ABB RobotStudio station: Glider program.rspag

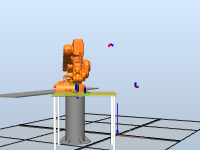
--- station ---
Station E459_norbert (saved by RobotStudio format 3)
Controller IRB140_6kg_0.81m_typeC_1, task T_ROB1: task frame (RAPID world) sits at (10, 680, 720) mm, rotated rx 0 ry 0 rz -30 deg in the station
Controller NorbertEGMVirtuel, task T_ROB1: task frame (RAPID world) sits at (-305, -752, 720) mm, rotated rx 0 ry 0 rz 30 deg in the station
Controller NorbertEGMVirtuel
  mechanical unit ROB_1: Norbert, 6 joints, base frame (0, 0, 0) mm
Controller IRB140_6kg_0.81m_typeC_1
  mechanical unit ROB_1: Rudolf, 6 joints, base frame (0, 0, 0) mm
Layout (positions relative to the parent item):
  - PedestalR [part, from Libraries\Pedestal.rslib] at (10, 680, 0) mm, rotated rx 0 ry 0 rz 150 deg
  - PedestalN [part, from Libraries\Pedestal.rslib] at (-305, -752, 0) mm, rotated rx 0 ry 0 rz -150 deg
  - Windowtable [part]
  - BordN [part, from Libraries\Desk.rslib] at (-421.89, -1050.54, 0) mm, rotated rx 0 ry 0 rz -60 deg
  - BordR [part, from Libraries\Desk.rslib] at (193.4, 1497.66, 0) mm, rotated rx 0 ry 0 rz -120 deg
  - UISpenholder [mechanism, from Libraries\UISpenholder.rslib] at (-60.57, -1074.38, 842.15) mm, rotated rx 179.64 ry 0.98 rz -67.17 deg
  - Norbert [mechanism, from Libraries\IRB140_6_81_C_01.rslib] at (-305, -752, 720) mm, rotated rx 0 ry 0 rz 30 deg; joint values [-1.4454, 0.9396, 0.5122, -0.0137, 0.1371, -2.8775] (rad or m)
  - Rudolf [mechanism, from Libraries\IRB140_6_81_C_01.rslib] at (10, 680, 720) mm, rotated rx 0 ry 0 rz -30 deg; joint values [1.249, 0.6446, -0.2193, 0, 1.1455, 1.249] (rad or m)
Attachment: BordN is attached to PedestalN
Attachment: BordR is attached to PedestalR
Attachment: UISpenholder is attached to Norbert / Link6
Station signals: DI doClose, DI doOpen
Station logic (signal -> signal, property => property):
  NorbertEGMVirtuel.doOpen -> ?.diOpen
  NorbertEGMVirtuel.doClose -> ?.diClose
  ?.doClosed -> NorbertEGMVirtuel.diClosed
Targets, tools, work objects and paths stored in the station and not in the controller backup, written as RAPID:
! task T_ROB1
MODULE EGM_test_UDP
  PROC testAO()
    SetAO ao_Joint1,0;
    SetAO ao_Joint2,0;
    SetAO ao_Joint3,0;
    SetAO ao_Joint4,0;
    SetAO ao_Joint5,0;
    SetAO ao_Joint6,0;
    MoveJ p20,v1000,fine,UISpenholder;
    SetAO ao_MoveX,0;
    SetAO ao_MoveY,0;
    SetAO ao_MoveZ,0;
  ENDPROC
ENDMODULE

! task T_ROB1
MODULE EGM_test_analog
  CONST jointtarget jpos10:=[[0,0,0,0,35,0],[9E9,9E9,9E9,9E9,9E9,9E9]];
  VAR signalao ao_MoveX;
  VAR signalao ao_MoveY;
  VAR signalao ao_MoveZ;
  TASK PERS loaddata load1:=[5,[0,1,0],[1,0,0,0],0,0,0];
  VAR signalao ao_RotX;
  VAR signalao ao_RotY;
  VAR signalao ao_RotZ;
ENDMODULE


--- Backups/IRB140_6kg_0.81m_typeC_1/RAPID/TASK1/PROGMOD/CalibData.mod ---
MODULE CalibData
	TASK PERS wobjdata WorkObj_Bord:=[FALSE,TRUE,"",[[194.800677646,-394.451457857,8],[1,0,0,0]],[[0,0,0],[1,0,0,0]]];


ENDMODULE

--- Backups/IRB140_6kg_0.81m_typeC_1/RAPID/TASK1/PROGMOD/EGMtest.mod ---
MODULE EGMtest
ENDMODULE

--- Backups/NorbertEGMVirtuel/RAPID/TASK1/PROGMOD/CalibData.mod ---
MODULE CalibData
ENDMODULE

--- Backups/NorbertEGMVirtuel/RAPID/TASK1/PROGMOD/EGM_test_UDP.mod ---
MODULE EGM_test_UDP

    VAR egmident egmID1;
    VAR egmstate egmSt1;

    CONST egm_minmax egm_minmax_lin1:=[-1,1]; !in mm
    CONST egm_minmax egm_minmax_rot1:=[-2,2];! in degees
    CONST robtarget p20:=[[34,-499,123],[0.000494947,0.662278052,-0.749217059,-0.007831731],[0,0,-1,0],[9E9,9E9,9E9,9E9,9E9,9E9]];

    PERS tooldata UISpenholder:=[TRUE,[[0,0,114.25],[1,0,0,0]],[1,[-0.095984607,0.082520613,38.69176324],[1,0,0,0],0,0,0]];
    TASK PERS wobjdata wobjBordN:=[FALSE,TRUE,"",[[0,0,0],[1,0,0,0]],[[150,-500,8],[0.707106781,0,0,-0.707106781]]];

    VAR pose posecorTable:=[[150,-500,8],[1,0,0,0]];
    VAR pose posesenTable:=[[0,0,0],[1,0,0,0]];

    PROC main()
        ! Move to start position. Fine point is demanded.
        MoveJ p20,v100,fine,UISpenholder;
        testuc_UDP;
    ENDPROC


    PROC testuc_UDP()
        EGMReset egmID1;
        EGMGetId egmID1;
        egmSt1 := EGMGetState(egmID1);
        TPWrite "EGM state: "\Num := egmSt1;

        IF egmSt1 <= EGM_STATE_CONNECTED THEN
            ! Set up the EGM data source: UdpUc server using device "EGMsensor:"and configuration "default"
            EGMSetupUC ROB_1, egmID1, "default", "EGMSensor:" \pose;
        ENDIF

        !Which program to run
        runEGM;


        IF egmSt1 = EGM_STATE_CONNECTED THEN
            TPWrite "Reset EGM instance egmID1";
            EGMReset egmID1;
        ENDIF
    ENDPROC


        PROC runEGM()
            EGMActPose egmID1\Tool:=UISpenholder \WObj:=wobj0, posecorTable,EGM_FRAME_WOBJ, posesenTable, EGM_FRAME_WOBJ
            \x:=egm_minmax_lin1 \y:=egm_minmax_lin1 \z:=egm_minmax_lin1
            \rx:=egm_minmax_rot1 \ry:=egm_minmax_rot1 \rz:=egm_minmax_rot1\LpFilter:=2\Samplerate:=4\MaxSpeedDeviation:= 1000;

            EGMRunPose egmID1, EGM_STOP_RAMP_DOWN\x \y \z\CondTime:=20 \RampInTime:=0.05\RampOutTime:=0.5;
            egmSt1:=EGMGetState(egmID1);
        ENDPROC

ENDMODULE

--- Backups/NorbertEGMVirtuel/RAPID/TASK1/SYSMOD/LINKEDM.sys ---
%%%
  VERSION:1
  LANGUAGE:ENGLISH
%%%

MODULE LINKEDM (SYSMODULE)

! FOLLOWER
!     Name of electronically linked follower axis used by operator at teach pendent.
      PERS string l_f_axis_name{5}       :=  ["",  "", "", "", ""];

!     Name of the mechanical unit for follower axis.
      PERS string l_f_mecunt_n{5}  :=  ["", "", "", "", ""];

!     Linked follower axis number in the mechanical unit (first axis in mech. unit is number 1).
      PERS num l_f_axis_no{5}      :=  [0,          0,   0,  0,  0];

! MASTER
!     Name of the mechanical unit for linked master axis.
      PERS string l_m_mecunt_n{5} :=  ["", "", "", "", ""];

!     Linked master axis number in the mechanical unit (first axis in mech. unit is number 1).
!     See axis number table in documentation for different master mechanical units.
      PERS num l_m_axis_no{5}     :=  [0,  0,  0,  0,  0];

! POSITION OFFSET
!     The increase of the allowed offset position between the master and follower
!     positions, used when starting AUTO mode. As soon as the offset is decreased
!     the old configurated parameter is used.
!     Example: 3 => the configurated value of allowed offset is increased 3 times.
      PERS num offset_ratio{5}       :=  [10,  10,   10,  10,  10];

! SPEED RATIO
!     Speed_ratio used in AUTO and JOG modes [ very_slow   slow    normal    fast]
!     Value 1 = max allowed manual speed.
      CONST num speed_ratio {20}      := [0.01, 0.01, 0.01, 0.01, 0.01,
                                          0.05, 0.05, 0.05, 0.05, 0.05,
                                          0.20, 0.20, 0.20, 0.20, 0.20,
                                          1.00, 1.00, 1.00, 1.00, 1.00];

! STEP SIZE
!     Displacement position used in JOG mode for each activation of positive or
!     negative movement.                  [very_short    short   normal   long]
!     Unit degees or meter.
      CONST num displacement {20}     := [0.001, 0.001, 0.001, 0.001, 0.001,
                                          0.005, 0.005, 0.005, 0.005, 0.005,
                                          0.020, 0.020, 0.020, 0.020, 0.020,
                                          0.100, 0.100, 0.100, 0.100, 0.100];


!-------------------------------------------------------------
 PROC Linked_m ()
      Linked_m_exe ;
 ENDPROC
ENDMODULE

--- Backups/IRB140_6kg_0.81m_typeC_1/SYSPAR/EIO.cfg ---
EIO:CFG_1.0:5:0::
#
EIO_BUS:

      -Name "Virtual1" -ConnectorID "SIM1"

      -Name "DeviceNet_Lean" -BusType "DNLE" -ConnectorID "PCI1"\
      -ConnectorLabel "DeviceNet Lean"
#
EIO_UNIT_TYPE:

      -Name "Virtual" -VendorName "ABB" -ProductName "Virtual unit"

      -Name "d651_Lean" -BusType "DNLE" -VendorName "ABB Robotics"\
      -ProductName "Combi Unit" -DL_ProductCode 25

      -Name "d652_Lean" -BusType "DNLE" -VendorName "ABB Robotics"\
      -ProductName "24 VDC Unit" -DL_ProductCode 26

      -Name "d653_Lean" -BusType "DNLE" -VendorName "ABB Robotics"\
      -ProductName "Relay Unit" -DL_ProductCode 27

      -Name "AC500_PLC_Lean" -BusType "DNLE" -VendorName "ABB Stotz"\
      -ProductName "AC500 PLC - FPB" -DL_ProductCode 1 -DL_VendorID 760

      -Name "DL_GENERIC" -BusType "DNLE" -DL_ProductCode 3535

      -Name "DL_GENERIC_POLL" -BusType "DNLE" -DL_ProductCode 3535\
      -DL_Pollrate 30

      -Name "d351_Lean" -BusType "DNLE" -VendorName "ABB Robotics"\
      -ProductName "IBS Adapter" -DL_ProductCode 7

      -Name "d378_Lean" -BusType "DNLE" -VendorName "ABB Robotics"\
      -ProductName "CCLink Adapter" -DL_ProductCode 17

      -Name "d377_Lean" -BusType "DNLE" -VendorName "ABB Robotics"\
      -ProductName "Qtracker" -DL_ProductCode 16 -DL_Pollrate 20
#
EIO_UNIT:

      -Name "Qtrack1" -UnitType "d377_Lean" -Bus "DeviceNet_Lean" -DL_Address 10

      -Name "DIGITAL_IO" -UnitType "d652_Lean" -Bus "DeviceNet_Lean"\
      -DL_Address 11
#
EIO_SIGNAL:

      -Name "c1Position" -SignalType "AI" -Unit "Qtrack1" -UnitMap "0-31"\
      -MaxLog 21474.8 -MaxPhys 1 -MaxPhysLimit 1 -MaxBitVal 2147483647\
      -MinLog -21474.8 -MinPhys -1 -MinPhysLimit -1 -MinBitVal -2147483647

      -Name "c1Speed" -SignalType "AI" -Unit "Qtrack1" -UnitMap "32-63"\
      -MaxLog 21474.8 -MaxPhys 1 -MaxPhysLimit 1 -MaxBitVal 2147483647\
      -MinLog -21474.8 -MinPhys -1 -MinPhysLimit -1 -MinBitVal -2147483647

      -Name "c1Connected" -SignalType "DI" -Unit "Qtrack1" -UnitMap "104"

      -Name "c1NullSpeed" -SignalType "DI" -Unit "Qtrack1" -UnitMap "105"

      -Name "c1DReady" -SignalType "DI" -Unit "Qtrack1" -UnitMap "106"

      -Name "c1PassStw" -SignalType "DI" -Unit "Qtrack1" -UnitMap "107"

      -Name "c1NewObjStrobe" -SignalType "DI" -Unit "Qtrack1" -UnitMap "108"

      -Name "c1EncSelected" -SignalType "DI" -Unit "Qtrack1" -UnitMap "109"

      -Name "c1EncAFautlt" -SignalType "DI" -Unit "Qtrack1" -UnitMap "110"

      -Name "c1EncBFautlt" -SignalType "DI" -Unit "Qtrack1" -UnitMap "111"

      -Name "c1Simulating" -SignalType "DI" -Unit "Qtrack1" -UnitMap "112"

      -Name "c1DirOfTravel" -SignalType "DI" -Unit "Qtrack1" -UnitMap "113"

      -Name "c1ScaleEncPuls" -SignalType "DI" -Unit "Qtrack1" -UnitMap "114"

      -Name "c1PowerUpStatus" -SignalType "DI" -Unit "Qtrack1" -UnitMap "83"

      -Name "c1WaitWObj" -SignalType "DO" -Unit "Qtrack1" -UnitMap "0"

      -Name "c1DropWObj" -SignalType "DO" -Unit "Qtrack1" -UnitMap "1"

      -Name "c1Rem1PObj" -SignalType "DO" -Unit "Qtrack1" -UnitMap "2"

      -Name "c1RemAllPObj" -SignalType "DO" -Unit "Qtrack1" -UnitMap "3"

      -Name "c1EncSelect" -SignalType "DO" -Unit "Qtrack1" -UnitMap "4"

      -Name "c1SoftSyncSig" -SignalType "DO" -Unit "Qtrack1" -UnitMap "5"

      -Name "c1SoftCheckSig" -SignalType "DO" -Unit "Qtrack1" -UnitMap "6"

      -Name "c1SimMode" -SignalType "DO" -Unit "Qtrack1" -UnitMap "7"

      -Name "c1CntToEncStr" -SignalType "DO" -Unit "Qtrack1" -UnitMap "40"

      -Name "c1ForceJob" -SignalType "DO" -Unit "Qtrack1" -UnitMap "41"

      -Name "c1PosInJobQ" -SignalType "DO" -Unit "Qtrack1" -UnitMap "42"

      -Name "c1ObjectsInQ" -SignalType "GI" -Unit "Qtrack1" -UnitMap "64-71"

      -Name "c1CntFromEnc1" -SignalType "GI" -Unit "Qtrack1" -UnitMap "72-87"

      -Name "c1CntFromEnc2" -SignalType "GI" -Unit "Qtrack1" -UnitMap "88-103"

      -Name "c1DTimestamp" -SignalType "GI" -Unit "Qtrack1" -UnitMap "120-151"

      -Name "c1CntToEnc1" -SignalType "GO" -Unit "Qtrack1" -UnitMap "8-23"

      -Name "c1CntToEnc2" -SignalType "GO" -Unit "Qtrack1" -UnitMap "24-39"

      -Name "GruppeUt" -SignalType "GO" -Unit "DIGITAL_IO" -UnitMap "0-7"\
      -Access "Default"

      -Name "GruppeInn" -SignalType "GI" -Unit "DIGITAL_IO" -UnitMap "0-7"\
      -Access "Default"

      -Name "LukkeGriper" -SignalType "DO" -Unit "DIGITAL_IO"\
      -SignalLabel "Lukke Griper" -UnitMap "9"

      -Name "Apnegriper" -SignalType "DO" -Unit "DIGITAL_IO"\
      -SignalLabel "Åpne griper" -UnitMap "8"
#
EIO_COMMAND:

      -Unit "Qtrack1" -CommandType "CountsPerMeter" -Value "10000.0"

      -Unit "Qtrack1" -CommandType "SyncSeparation" -Value "0.005"

      -Unit "Qtrack1" -CommandType "QueueTrckDist" -Value "0.0"

      -Unit "Qtrack1" -CommandType "StartWinWidth" -Value "10.0"

      -Unit "Qtrack1" -CommandType "IIRFPeriod" -Value "0.02"

      -Unit "Qtrack1" -CommandType "IIRFNoOfPoles" -Value "2"

      -Unit "Qtrack1" -CommandType "IIRFNoOfZeroes" -Value "0"

      -Unit "Qtrack1" -CommandType "IIRFXfrmMetPol" -Value "1"

      -Unit "Qtrack1" -CommandType "IIRFXfrmMetZero" -Value "1"

      -Unit "Qtrack1" -CommandType "IIRFFZ" -Value "0.0"

      -Unit "Qtrack1" -CommandType "IIRFDZ" -Value "0.0"

      -Unit "Qtrack1" -CommandType "IIRFFP" -Value "2.0"

      -Unit "Qtrack1" -CommandType "IIRFDP" -Value "0.707"

      -Unit "Qtrack1" -CommandType "IIRFGain" -Value "1.0"

      -Unit "Qtrack1" -CommandType "FIRFLength" -Value "0"

      -Unit "Qtrack1" -CommandType "FIRFB0" -Value "0.0"

      -Unit "Qtrack1" -CommandType "FIRFB1" -Value "0.0"

      -Unit "Qtrack1" -CommandType "AutoBackup" -Value "1"

      -Unit "Qtrack1" -CommandType "SimulationVel" -Value "0.100"

      -Unit "Qtrack1" -CommandType "ScalingFactor" -Value "100.0"

      -Unit "Qtrack1" -CommandType "CheckPointDist" -Value "0.0"

      -Unit "Qtrack1" -CommandType "CheckPWinWidth" -Value "0.0"
#
EIO_COMMAND_TYPE:

      -Name "StationNo_L" -UnitType "d378_Lean" -DefValue "1" -OrderNr 1\
      -DL_Path "6,20 68 24 01 30 01,C6,1"

      -Name "BaudRate_L" -UnitType "d378_Lean" -DefValue "0" -OrderNr 2\
      -DL_Path "6,20 68 24 01 30 02,C6,1"

      -Name "OccStat_L" -UnitType "d378_Lean" -DefValue "1" -OrderNr 3\
      -DL_Path "6,20 68 24 01 30 03,C6,1"

      -Name "BasicIO_L" -UnitType "d378_Lean" -DefValue "0" -OrderNr 4\
      -DL_Path "6,20 68 24 01 30 04,C1,1"

      -Name "D378reset_L" -UnitType "d378_Lean" -DefValue "0" -OrderNr 5\
      -DL_Path "4,20 01 24 01,C1,1" -DL_Service 5

      -Name "DataWidth_L" -UnitType "d351_Lean" -DefValue "3" -OrderNr 1\
      -DL_Path "6,20 65 24 01 30 01,C6,1"

      -Name "D351reset_L" -UnitType "d351_Lean" -DefValue "0" -OrderNr 2\
      -DL_Path "4,20 01 24 01,C1,1" -DL_Service 5

      -Name "CountsPerMeter" -UnitType "d377_Lean" -DefValue "10000.0"\
      -OrderNr 2 -DL_Path "6,20 66 24 01 30 01,CA,4"

      -Name "SyncSeparation" -UnitType "d377_Lean" -DefValue "0.1" -OrderNr 3\
      -DL_Path "6,20 66 24 01 30 02,CA,4"

      -Name "QueueTrckDist" -UnitType "d377_Lean" -DefValue "0.0" -OrderNr 4\
      -DL_Path "6,20 66 24 01 30 03,CA,4"

      -Name "StartWinWidth" -UnitType "d377_Lean" -DefValue "0.5" -OrderNr 5\
      -DL_Path "6,20 66 24 01 30 04,CA,4"

      -Name "AutoBackup" -UnitType "d377_Lean" -DefValue "1" -OrderNr 6\
      -DL_Path "6,20 66 24 01 30 12,C1,1"

      -Name "SimulationVel" -UnitType "d377_Lean" -DefValue "0.1" -OrderNr 7\
      -DL_Path "6,20 66 24 01 30 13,CA,4"

      -Name "ScalingFactor" -UnitType "d377_Lean" -DefValue "100" -OrderNr 8\
      -DL_Path "6,20 66 24 01 30 14,CA,4"

      -Name "CheckPointDist" -UnitType "d377_Lean" -DefValue "0.0" -OrderNr 9\
      -DL_Path "6,20 66 24 01 30 15,CA,4"

      -Name "CheckPWinWidth" -UnitType "d377_Lean" -DefValue "0.0" -OrderNr 10\
      -DL_Path "6,20 66 24 01 30 16,CA,4"

      -Name "IIRFPeriod" -UnitType "d377_Lean" -DefValue "0.02" -OrderNr 11\
      -DL_Path "6,20 66 24 01 30 05,CA,4"

      -Name "IIRFNoOfPoles" -UnitType "d377_Lean" -DefValue "2" -OrderNr 12\
      -DL_Path "6,20 66 24 01 30 06,C6,1"

      -Name "IIRFNoOfZeroes" -UnitType "d377_Lean" -DefValue "0" -OrderNr 13\
      -DL_Path "6,20 66 24 01 30 07,C6,1"

      -Name "IIRFXfrmMetPol" -UnitType "d377_Lean" -DefValue "1" -OrderNr 14\
      -DL_Path "6,20 66 24 01 30 08,C6,1"

      -Name "IIRFXfrmMetZero" -UnitType "d377_Lean" -DefValue "1" -OrderNr 15\
      -DL_Path "6,20 66 24 01 30 09,C6,1"

      -Name "IIRFFZ" -UnitType "d377_Lean" -DefValue "0.0" -OrderNr 16\
      -DL_Path "6,20 66 24 01 30 0A,CA,4"

      -Name "IIRFDZ" -UnitType "d377_Lean" -DefValue "0.0" -OrderNr 17\
      -DL_Path "6,20 66 24 01 30 0B,CA,4"

      -Name "IIRFFP" -UnitType "d377_Lean" -DefValue "2.0" -OrderNr 18\
      -DL_Path "6,20 66 24 01 30 0C,CA,4"

      -Name "IIRFDP" -UnitType "d377_Lean" -DefValue "0.707" -OrderNr 19\
      -DL_Path "6,20 66 24 01 30 0D,CA,4"

      -Name "IIRFGain" -UnitType "d377_Lean" -DefValue "1.0" -OrderNr 20\
      -DL_Path "6,20 66 24 01 30 0E,CA,4"

      -Name "FIRFLength" -UnitType "d377_Lean" -DefValue "1" -OrderNr 21\
      -DL_Path "6,20 66 24 01 30 0F,C6,1"

      -Name "FIRFB0" -UnitType "d377_Lean" -DefValue "0.0" -OrderNr 22\
      -DL_Path "6,20 66 24 01 30 10,CA,4"

      -Name "FIRFB1" -UnitType "d377_Lean" -DefValue "0.0" -OrderNr 23\
      -DL_Path "6,20 66 24 01 30 11,CA,4"

      -Name "TimeKeeperInit" -UnitType "d377_Lean" -DefValue "0" -OrderNr 1\
      -DL_Path "6,20 68 24 01 30 01,C1,1"
#
EIO_ACCESS:

      -Name "All" -Rapid  -LocalManual  -LocalAuto  -RemoteManual  -RemoteAuto

--- Backups/NorbertEGMVirtuel/SYSPAR/EIO.cfg ---
EIO:CFG_1.0:6:1::
#
INDUSTRIAL_NETWORK:

      -Name "DeviceNet" -Label "DeviceNet Master/Slave Network" -Address "2"

      -Name "DeviceNet_Anybus" -Label "DeviceNet Anybus Network" -Address "20"
#
DEVICENET_DEVICE:

      -Name "Qtrack1" -Simulated  -VendorName "ABB Robotics"\
      -ProductName "Qtracker" -Address 15 -ProductCode 16 -DeviceType 100\
      -PollRate 20 -OutputSize 6 -InputSize 19

      -Name "DIGITAL_IO" -VendorName "ABB Robotics"\
      -ProductName "24 VDC I/O Device" -Label "DSQC 652 24 VDC I/O Device"\
      -Address 11 -ProductCode 26 -DeviceType 7 -ConnectionType "COS"\
      -OutputSize 2 -InputSize 2
#
DEVICENET_DEVICE_TEMPLATE:

      -Name "d377B" -VendorName "ABB Robotics" -ProductName "Qtracker"\
      -Label "DSQC 377B Queue Tracker" -ProductCode 16 -DeviceType 100\
      -PollRate 20 -OutputSize 6 -InputSize 19
#
DEVICENET_COMMAND:

      -Name "CountsPerMeter1" -Device "Qtrack1" -OrderNr 2\
      -Path "6,20 66 24 01 30 01,CA,4" -Value "20000.0"

      -Name "SyncSeparation1" -Device "Qtrack1" -OrderNr 3\
      -Path "6,20 66 24 01 30 02,CA,4" -Value "0.005"

      -Name "QueueTrckDist1" -Device "Qtrack1" -OrderNr 4\
      -Path "6,20 66 24 01 30 03,CA,4" -Value "0.0"

      -Name "StartWinWidth1" -Device "Qtrack1" -OrderNr 5\
      -Path "6,20 66 24 01 30 04,CA,4" -Value "10.0"

      -Name "AutoBackup1" -Device "Qtrack1" -OrderNr 6\
      -Path "6,20 66 24 01 30 12,C1,1" -Value "1"

      -Name "SimulationVel1" -Device "Qtrack1" -OrderNr 7\
      -Path "6,20 66 24 01 30 13,CA,4" -Value "0.100"

      -Name "ScalingFactor1" -Device "Qtrack1" -OrderNr 8\
      -Path "6,20 66 24 01 30 14,CA,4" -Value "2000.0"

      -Name "CheckPointDist1" -Device "Qtrack1" -OrderNr 9\
      -Path "6,20 66 24 01 30 15,CA,4" -Value "0.0"

      -Name "CheckPWinWidth1" -Device "Qtrack1" -OrderNr 10\
      -Path "6,20 66 24 01 30 16,CA,4" -Value "0.0"

      -Name "IIRFPeriod1" -Device "Qtrack1" -OrderNr 11\
      -Path "6,20 66 24 01 30 05,CA,4" -Value "0.02"

      -Name "IIRFNoOfPoles1" -Device "Qtrack1" -OrderNr 12\
      -Path "6,20 66 24 01 30 06,C6,1" -Value "2"

      -Name "IIRFNoOfZeroes1" -Device "Qtrack1" -OrderNr 13\
      -Path "6,20 66 24 01 30 07,C6,1" -Value "0"

      -Name "IIRFXfrmMetPol1" -Device "Qtrack1" -OrderNr 14\
      -Path "6,20 66 24 01 30 08,C6,1" -Value "1"

      -Name "IIRFXfrmMetZero1" -Device "Qtrack1" -OrderNr 15\
      -Path "6,20 66 24 01 30 09,C6,1" -Value "1"

      -Name "IIRFFZ1" -Device "Qtrack1" -OrderNr 16\
      -Path "6,20 66 24 01 30 0A,CA,4" -Value "0.0"

      -Name "IIRFDZ1" -Device "Qtrack1" -OrderNr 17\
      -Path "6,20 66 24 01 30 0B,CA,4" -Value "0.0"

      -Name "IIRFFP1" -Device "Qtrack1" -OrderNr 18\
      -Path "6,20 66 24 01 30 0C,CA,4" -Value "2.0"

      -Name "IIRFDP1" -Device "Qtrack1" -OrderNr 19\
      -Path "6,20 66 24 01 30 0D,CA,4" -Value "0.707"

      -Name "IIRFGain1" -Device "Qtrack1" -OrderNr 20\
      -Path "6,20 66 24 01 30 0E,CA,4" -Value "1.0"

      -Name "FIRFLength1" -Device "Qtrack1" -OrderNr 21\
      -Path "6,20 66 24 01 30 0F,C6,1" -Value "0"

      -Name "FIRFB01" -Device "Qtrack1" -OrderNr 22\
      -Path "6,20 66 24 01 30 10,CA,4" -Value "0.0"

      -Name "FIRFB11" -Device "Qtrack1" -OrderNr 23\
      -Path "6,20 66 24 01 30 11,CA,4" -Value "0.0"
#
DEVICENET_INTERNAL_DEVICE:

      -Name "DN_Internal_Device" -VendorName "ABB Robotics"\
      -ProductName "DeviceNet Internal Slave Device"
#
DEVICENET_INTERNAL_ANYBUS_DEVICE:

      -Name "DN_Internal_Anybus" -VendorName "ABB Robotics"\
      -ProductName "DeviceNet Internal Anybus Slave Device"
#
EIO_SIGNAL:

      -Name "c1Position" -SignalType "AI" -Device "Qtrack1" -DeviceMap "0-31"\
      -MaxLog 21474.8 -MaxPhys 1 -MaxPhysLimit 1 -MaxBitVal 2147483647\
      -MinLog -21474.8 -MinPhys -1 -MinPhysLimit -1 -MinBitVal -2147483647

      -Name "c1Speed" -SignalType "AI" -Device "Qtrack1" -DeviceMap "32-63"\
      -MaxLog 21474.8 -MaxPhys 1 -MaxPhysLimit 1 -MaxBitVal 2147483647\
      -MinLog -21474.8 -MinPhys -1 -MinPhysLimit -1 -MinBitVal -2147483647

      -Name "c1Connected" -SignalType "DI" -Device "Qtrack1" -DeviceMap "104"

      -Name "c1NullSpeed" -SignalType "DI" -Device "Qtrack1" -DeviceMap "105"

      -Name "c1DReady" -SignalType "DI" -Device "Qtrack1" -DeviceMap "106"

      -Name "c1PassStw" -SignalType "DI" -Device "Qtrack1" -DeviceMap "107"

      -Name "c1NewObjStrobe" -SignalType "DI" -Device "Qtrack1" -DeviceMap "108"

      -Name "c1EncSelected" -SignalType "DI" -Device "Qtrack1" -DeviceMap "109"

      -Name "c1EncAFautlt" -SignalType "DI" -Device "Qtrack1" -DeviceMap "110"

      -Name "c1EncBFautlt" -SignalType "DI" -Device "Qtrack1" -DeviceMap "111"

      -Name "c1Simulating" -SignalType "DI" -Device "Qtrack1" -DeviceMap "112"

      -Name "c1DirOfTravel" -SignalType "DI" -Device "Qtrack1" -DeviceMap "113"

      -Name "c1ScaleEncPuls" -SignalType "DI" -Device "Qtrack1" -DeviceMap "114"

      -Name "c1PowerUpStatus" -SignalType "DI" -Device "Qtrack1" -DeviceMap "83"

      -Name "c1WaitWObj" -SignalType "DO" -Device "Qtrack1" -DeviceMap "0"

      -Name "c1DropWObj" -SignalType "DO" -Device "Qtrack1" -DeviceMap "1"

      -Name "c1Rem1PObj" -SignalType "DO" -Device "Qtrack1" -DeviceMap "2"

      -Name "c1RemAllPObj" -SignalType "DO" -Device "Qtrack1" -DeviceMap "3"

      -Name "c1EncSelect" -SignalType "DO" -Device "Qtrack1" -DeviceMap "4"

      -Name "c1SoftSyncSig" -SignalType "DO" -Device "Qtrack1" -DeviceMap "5"

      -Name "c1SoftCheckSig" -SignalType "DO" -Device "Qtrack1" -DeviceMap "6"

      -Name "c1SimMode" -SignalType "DO" -Device "Qtrack1" -DeviceMap "7"

      -Name "c1CntToEncStr" -SignalType "DO" -Device "Qtrack1" -DeviceMap "40"

      -Name "c1ForceJob" -SignalType "DO" -Device "Qtrack1" -DeviceMap "41"

      -Name "c1PosInJobQ" -SignalType "DO" -Device "Qtrack1" -DeviceMap "42"

      -Name "c1ObjectsInQ" -SignalType "GI" -Device "Qtrack1" -DeviceMap "64-71"

      -Name "c1CntFromEnc" -SignalType "GI" -Device "Qtrack1"\
      -DeviceMap "72-103"

      -Name "c1DTimestamp" -SignalType "GI" -Device "Qtrack1"\
      -DeviceMap "120-151"

      -Name "c1CntToEnc" -SignalType "GO" -Device "Qtrack1" -DeviceMap "8-39"

      -Name "doGripOpen" -SignalType "DO" -Device "DIGITAL_IO"\
      -Label "Pneumatic gripper OPEN" -DeviceMap "9"

      -Name "doGripClose" -SignalType "DO" -Device "DIGITAL_IO"\
      -Label "Pneumatic gripper CLOSE" -DeviceMap "8"

      -Name "ao_Joint1" -SignalType "AO" -Device "Qtrack1" -DeviceMap "16-31"\
      -Access "All" -MaxLog 21474.8 -MaxPhys 500 -MaxPhysLimit 500\
      -MaxBitVal 32767 -MinLog -21474.8 -MinPhys -500 -MinPhysLimit -500\
      -MinBitVal -32767

      -Name "ao_Joint2" -SignalType "AO" -Device "Qtrack1" -DeviceMap "32-47"\
      -MaxLog 21474.8 -MaxPhys 500 -MaxPhysLimit 500 -MaxBitVal 32767\
      -MinLog -21474.8 -MinPhys -500 -MinPhysLimit -500 -MinBitVal -32767

      -Name "ao_Joint3" -SignalType "AO" -Device "Qtrack1" -DeviceMap "48-63"\
      -MaxLog 21474.8 -MaxPhys 500 -MaxPhysLimit 500 -MaxBitVal 32767\
      -MinLog -21474.8 -MinPhys -500 -MinPhysLimit -500 -MinBitVal -32767

      -Name "ao_Joint6" -SignalType "AO" -Device "Qtrack1" -DeviceMap "96-111"\
      -MaxLog 21474.8 -MaxPhys 500 -MaxPhysLimit 500 -MaxBitVal 32767\
      -MinLog -21474.8 -MinPhys -500 -MinPhysLimit -500 -MinBitVal -32767

      -Name "ao_Joint5" -SignalType "AO" -Device "Qtrack1" -DeviceMap "80-95"\
      -MaxLog 21474.8 -MaxPhys 500 -MaxPhysLimit 500 -MaxBitVal 32767\
      -MinLog -21474.8 -MinPhys -500 -MinPhysLimit -500 -MinBitVal -32767

      -Name "ao_Joint4" -SignalType "AO" -Device "Qtrack1" -DeviceMap "64-79"\
      -MaxLog 21474.8 -MaxPhys 500 -MaxPhysLimit 500 -MaxBitVal 32767\
      -MinLog -21474.8 -MinPhys -500 -MinPhysLimit -500 -MinBitVal -32767

      -Name "ao_MoveX" -SignalType "AO" -Device "Qtrack1" -DeviceMap "112-127"\
      -MaxLog 2147.8 -MaxPhys 500 -MaxPhysLimit 500 -MaxBitVal 32767\
      -MinLog -2147.8 -MinPhys -500 -MinPhysLimit -500 -MinBitVal -32767

      -Name "ao_MoveY" -SignalType "AO" -Device "Qtrack1" -DeviceMap "128-143"\
      -MaxLog 21474.8 -MaxPhys 500 -MaxPhysLimit 500 -MaxBitVal 32767\
      -MinLog -21474.8 -MinPhys -500 -MinPhysLimit -500 -MinBitVal -32767

      -Name "ao_MoveZ" -SignalType "AO" -Device "Qtrack1" -DeviceMap "144-159"\
      -MaxLog 21474.8 -MaxPhys 500 -MaxPhysLimit 500 -MaxBitVal 32767\
      -MinLog -21474.8 -MinPhys -500 -MinPhysLimit -500 -MinBitVal -32767

      -Name "ao_RotX" -SignalType "AO" -Device "Qtrack1" -DeviceMap "160-175"\
      -MaxLog 21474.8 -MaxPhys 500 -MaxPhysLimit 500 -MaxBitVal 32767\
      -MinLog -21474.8 -MinPhys -500 -MinPhysLimit -500 -MinBitVal -32767

      -Name "ao_RotY" -SignalType "AO" -Device "Qtrack1" -DeviceMap "176-191"\
      -MaxLog 21474.8 -MaxPhys 500 -MaxPhysLimit 500 -MaxBitVal 32767\
      -MinLog -21474.8 -MinPhys -500 -MinPhysLimit -500 -MinBitVal -32767

      -Name "ao_RotZ" -SignalType "AO" -Device "Qtrack1" -DeviceMap "192-207"\
      -MaxLog 21474.8 -MaxPhys 500 -MaxPhysLimit 500 -MaxBitVal 32767\
      -MinLog -21474.8 -MinPhys -500 -MinPhysLimit -500 -MinBitVal -32767

--- Backups/NorbertEGMVirtuel/SYSPAR/PROC.cfg ---
PROC:CFG_1.0:6:0::
#
CONVEYOR:

      -name "CNV1" -sensor_type "CAN" -use_sensor "CAN1" -adjustment_speed 850\
      -min_dist -600 -max_dist 20000 -correction_vector_ramp_length 5
#
CONVEYOR_CAN_SENSOR:

      -name "CAN1" -eio_unit_name "Qtrack1" -connected_signal "c1Connected"\
      -position_signal "c1Position" -velocity_signal "c1Speed"\
      -null_speed_signal "c1NullSpeed" -wait_wobj_signal "c1WaitWObj"\
      -drop_wobj_signal "c1DropWObj" -data_timestamp "c1DTimestamp"\
      -rem_all_pobj_signal "c1RemAllPObj" -rem_one_pobj_signal "c1Rem1PObj"\
      -supervise_max_dist_off  -newobj_strobe "c1NewObjStrobe"\
      -encA_fault_signal "c1EncAFautlt" -dir_of_travel_signal "c1DirOfTravel"\
      -force_job_signal "c1ForceJob" -count_to_enc_strobe "c1CntToEncStr"\
      -pos_in_jobq_signal "c1PosInJobQ" -obj_in_queue_signal "c1ObjectsInQ"\
      -count_from_enc "c1CntFromEnc" -count_to_enc "c1CntToEnc"\
      -scale_enc_puls "c1ScaleEncPuls"
